FUNCTION_BLOCK SM_TransferLine EXTENDS StateMachine
VAR_INPUT CONSTANT
	sTLMqttName : STRING(8);
END_VAR
VAR_OUTPUT
END_VAR
VAR
	
	aRollerConveyors : ARRAY[1..3] OF RollerConveyor;
	fbChainController : FB_ChainController;
	
	fbPalletizer : SM_Palletizer;
	fbStepWorkerReady : FB_StepWorker;
	fbStepWorkerBusy : FB_StepWorker;

	scBeltConveyors : 
		SC_BeltConveyors := 
		(
			sChainName  := 'scBeltConveyors',
			rChainController := fbChainController
		);
		
	scPostPalletizer : 
		SC_PostPalletizer := 
		(
			sChainName  := 'scPostPalletizer',
			rChainController := fbChainController
		);
		
	scPrePalletizer : 
		SC_PrePalletizer := 
		(
			sChainName  := 'scPrePalletizer',
			rChainController := fbChainController
		);
 
	uiPackageCounter : UINT;
	i : UINT;
	bPackageOnTheWay : BOOL;
	
END_VAR

SUPER^();
fbPalletizer(ioChainController := fbChainController);
scBeltConveyors(bAllPartsPresent := fbPalletizer.bAllPartsPresent);
scPrePalletizer();
scPrePalletizer.bPalletizerRequest := fbPalletizer.scFirstFloor.bPalletizerRequest;
fbPalletizer.scFirstFloor.bIncomingPallet := scPrePalletizer.bSentToPalletizer;
scPostPalletizer(sTLMqttName := sTLMqttName);

METHOD PROTECTED Busy : BOOL
VAR_INPUT
END_VAR
CASE fbStepWorkerBusy.uiStep OF
	eTlStartUnits:
		scBeltConveyors.bExecute := TRUE;
		scPrePalletizer.bExecute := TRUE;
		scPostPalletizer.bExecute := TRUE;
		fbPalletizer.bExecute := TRUE;
		fbStepWorkerBusy.mNextStep(eTlCheckUnits);
	eTlCheckUnits:
		IF scBeltConveyors.eStateMachine = E_StateMachine.eError
		THEN
			fbStepWorkerBusy.mNextStep(eTlSignalError);
		END_IF
	eTlSignalError:
		Fault();
END_CASE
END_METHOD

METHOD PROTECTED  Error : BOOL
VAR_INPUT
END_VAR
END_METHOD

METHOD PROTECTED  Idle : BOOL
VAR_INPUT
END_VAR
Start();
END_METHOD

METHOD PROTECTED  Init : BOOL
VAR_INPUT
END_VAR
fbChainController
	.addChain(itfChain := scBeltConveyors)
	.addChain(itfChain := scPostPalletizer)
	.addChain(itfChain := scPrePalletizer);
	
	
Start();
END_METHOD

METHOD PROTECTED  Prepare : BOOL
VAR_INPUT
END_VAR
END_METHOD

METHOD PROTECTED  Ready : BOOL
VAR_INPUT
END_VAR
END_METHOD

METHOD PROTECTED  Waiting : BOOL
VAR_INPUT
END_VAR
END_METHOD

END_FUNCTION_BLOCK

(* stored: Version 1.1.0.1, ProductVersion 3.1.4024.2
   POU SM_TransferLine: Id {6f843e77-bb22-480b-8b14-188352f305ee}, SpecialFunc None
   Method Busy: Id {ba0ee649-e6ac-40a4-ac17-f140d3419283}
   Method Error: Id {25dafad4-832a-4b58-a247-fab5222968c3}
   Method Idle: Id {f1f51908-c198-4971-a94a-ecbcd2e14002}
   Method Init: Id {b268c93a-f267-4f9d-9c0b-502444e4de54}
   Method Prepare: Id {c71298a5-214a-4fbd-bc50-6a1ff0be19ce}
   Method Ready: Id {b730c8ee-8bb5-459b-84c3-d41d010e0e7c}
   Method Waiting: Id {a1e703a8-39c7-4d9d-a5f5-59ed24c6ef8d} *)
